(* Logix 5000 project; controller optix_aio_sample 1756-L85E rev 35.11; software revision 35.00 *)

TASK MainTask (continuous, watchdog 500 ms) : MainProgram

MODULES
   Local : 1756-L85E (ICP 5, rev 35.11)
END_MODULES

VAR_GLOBAL   (* controller tags *)
   counter_tag : DINT;
END_VAR

PROGRAM MainProgram   (* main routine MainRoutine *)
VAR
   counter1 : COUNTER := (PRE := 1000);
   start : BOOL;
   timer1 : TIMER := (PRE := 1000);
END_VAR

ROUTINE MainRoutine   (* ladder *)
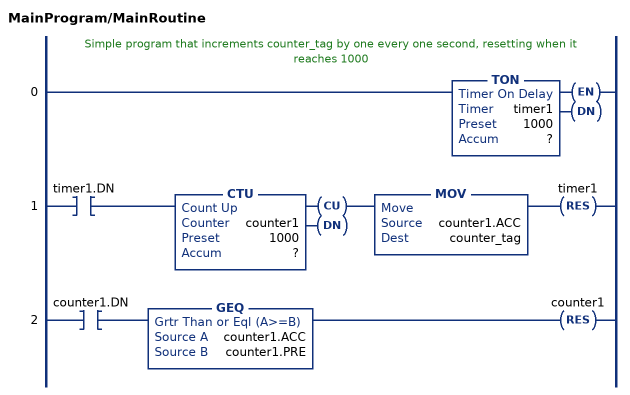
   // Simple program that increments counter_tag by one every one second, resetting when it reaches 1000
   0: TON(timer1,?,?);
   1: XIC(timer1.DN)CTU(counter1,?,?)MOV(counter1.ACC,counter_tag)RES(timer1);
   2: XIC(counter1.DN)GEQ(counter1.ACC,counter1.PRE)RES(counter1);
END_ROUTINE
END_PROGRAM
